FUNCTION_BLOCK THRESHOLD
  {SET_ATTRIBUTE(OpcUa, DEVICE.SENSOR)}
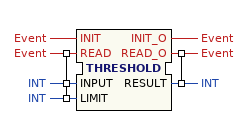
  EVENT_INPUT
    INIT;
    READ WITH INPUT, LIMIT;
  END_EVENT
  EVENT_OUTPUT
    INIT_O;
    READ_O WITH RESULT;
  END_EVENT
  VAR_INPUT
    INPUT : INT; {SET_ATTRIBUTE(OpcUa, Variable.RUN)}
    LIMIT : INT; {SET_ATTRIBUTE(OpcUa, Variable.RUN)}
  END_VAR
  VAR_OUTPUT
    RESULT : INT; {SET_ATTRIBUTE(OpcUa, Variable.RUN)}
  END_VAR
END_FUNCTION_BLOCK
